FUNCTION_BLOCK PIDBase_HMI (* Service Interface Function Block Type *)
  (* Standard: 61499-2 *)
  (* Version 1.0.1, 10/18/2023, ApplicationLibDevTeam, Schneider Electric, First Version *)
  PACKAGE Main;
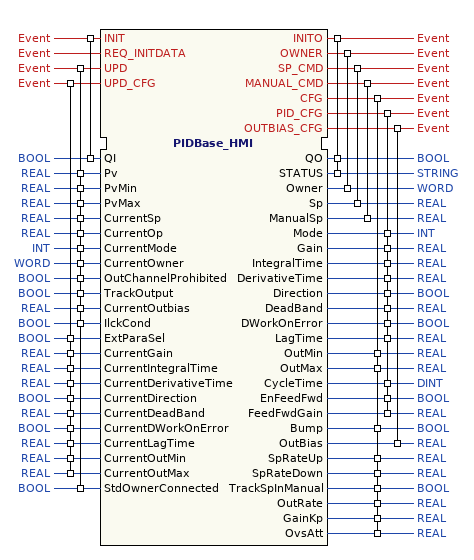
  EVENT_INPUT
    INIT WITH QI;
    REQ_INITDATA; (* Request to initialize data *)
    UPD WITH Pv, PvMin, PvMax, CurrentSp, CurrentOp, CurrentMode, OutChannelProhibited, TrackOutput, CurrentOutbias, IlckCond, StdOwnerConnected, CurrentOwner; (* Update data to supervision *)
    UPD_CFG WITH ExtParaSel, CurrentGain, CurrentIntegralTime, CurrentDerivativeTime, CurrentLagTime, CurrentDeadBand, CurrentOutMin, CurrentOutMax, CurrentDWorkOnError, CurrentDirection; (* Update external parameter data to supervision *)
  END_EVENT
  EVENT_OUTPUT
    INITO WITH QO, STATUS;
    OWNER WITH Owner; (* Request for owner change *)
    SP_CMD WITH Sp; (* Request to update operator setpoint in auto mode *)
    MANUAL_CMD WITH ManualSp; (* Request to update operator setpoint in manual mode *)
    CFG WITH OutMin, OutMax, Bump, SpRateUp, SpRateDown, TrackSpInManual, OutRate, GainKp, OvsAtt; (* Request to update generic parameters *)
    PID_CFG WITH Gain, DerivativeTime, IntegralTime, Mode, LagTime, DeadBand, Direction, CycleTime, DWorkOnError, EnFeedFwd, FeedFwdGain; (* Request to update PID parameter *)
    OUTBIAS_CFG WITH OutBias; (* Request to update outbias configuration *)
  END_EVENT
  VAR_INPUT
    QI : BOOL;
    Pv : REAL; (* Process value *) {SET_ATTRIBUTE(Runtime.Archive.Counters, AbsoluteValues=False)} {SET_ATTRIBUTE(Runtime.Archive.Id, 1)} {SET_ATTRIBUTE(Runtime.History.Depth, 500)} {SET_ATTRIBUTE(Runtime.History.SmoothTime, 60000)} {SET_ATTRIBUTE(Runtime.History.SmoothValue, 0.1)}
    PvMin : REAL; (* Minimum range of process value *)
    PvMax : REAL; (* Maximum range of process value *)
    CurrentSp : REAL; (* Current setpoint value *) {SET_ATTRIBUTE(Runtime.Archive.Counters, AbsoluteValues=False)} {SET_ATTRIBUTE(Runtime.Archive.Id, 1)} {SET_ATTRIBUTE(Runtime.History.Depth, 500)} {SET_ATTRIBUTE(Runtime.History.SmoothTime, 60000)} {SET_ATTRIBUTE(Runtime.History.SmoothValue, 0.1)}
    CurrentOp : REAL; (* Current output value *) {SET_ATTRIBUTE(Runtime.Archive.Counters, AbsoluteValues=False)} {SET_ATTRIBUTE(Runtime.Archive.Id, 1)} {SET_ATTRIBUTE(Runtime.History.Depth, 500)} {SET_ATTRIBUTE(Runtime.History.SmoothTime, 60000)} {SET_ATTRIBUTE(Runtime.History.SmoothValue, 0.1)}
    CurrentMode : INT; (* Current mode selected *)
    CurrentOwner : WORD; (* Current Owner status *)
    OutChannelProhibited : BOOL; (* 1 = Output change prohibited *)
    TrackOutput : BOOL; (* 1 = Output tracking active *)
    CurrentOutbias : REAL; (* Current ouput bias value *)
    IlckCond : BOOL; (* 1= Interlock active *)
    ExtParaSel : BOOL; (* 1 = External paramters available for PID calculation *)
    CurrentGain : REAL; (* Current gain for PID calculation *)
    CurrentIntegralTime : REAL; (* Current integral time for PID calculation *)
    CurrentDerivativeTime : REAL; (* Current derivative time for PID calculation *)
    CurrentDirection : BOOL; (* Current direction of PID calculation *)
    CurrentDeadBand : REAL; (* Current deadband for PID calculation *)
    CurrentDWorkOnError : BOOL; (* Current derivative work on error for PID calculation *)
    CurrentLagTime : REAL; (* Current lagtime for PID calculation *)
    CurrentOutMin : REAL; (* Current minimum ouput value for PID calculation *)
    CurrentOutMax : REAL; (* Current maximum ouput value for PID calculation *)
    StdOwnerConnected : BOOL; (* 1= External owner connected *)
  END_VAR
  VAR_OUTPUT
    QO : BOOL; (* Event Output Qualifier *)
    STATUS : STRING; (* Service Status *)
    Owner : WORD; (* Requested owner (16#10 = Operator, 16#8 = Program remote) *)
    Sp : REAL; (* Setpoint for PID calculation *)
    ManualSp : REAL; (* Manual setpoint for PID calculation *)
    Mode : INT; (* Mode for PID calculation (0 = Manual Mode, 1 = Auto Mode) *)
    Gain : REAL; (* Gain parameter for P calculation *)
    IntegralTime : REAL; (* Gain parameter for I calculation *)
    DerivativeTime : REAL; (* Parameter for D calculation *)
    Direction : BOOL; (* Direction for error calculation (0 = Pv-Sp; 1 = Sp-Pv) *)
    DeadBand : REAL; (* Deadband for I and D calculation *)
    DWorkOnError : BOOL; (* 1 = D work on error; 0 = D work on Pv *)
    LagTime : REAL; (* Lag time parameter for D calculation *)
    OutMin : REAL; (* Minimum range of ouput value *)
    OutMax : REAL; (* Maximum range of ouput value *)
    CycleTime : DINT; (* Cycletime for PID calculation (ms) *)
    EnFeedFwd : BOOL; (* 1 = Feedforward active *)
    FeedFwdGain : REAL; (* Feed forward gain value *)
    Bump : BOOL; (* 1 =Transition to automatic mode with bump ,0= Bumpless transition to automatic mode *)
    OutBias : REAL; (* Output offset (bias) value in Auto Mode and Integration time is zero *)
    SpRateUp : REAL; (* Setpoint rate to move up *)
    SpRateDown : REAL; (* Setpoint rate to move down *)
    TrackSpInManual : BOOL; (* 1 = Sp tracking to Pv is enabled in manual mode *)
    OutRate : REAL; (* Limit for output modification in units per second (≥ 0) *)
    GainKp : REAL; (* Reducing the proportional contribution within the dead zone dband *)
    OvsAtt : REAL; (* Reducing the overrun ( Should be between 0  to 1) *)
  END_VAR
  SERVICE /
    SEQUENCE 
    END_SEQUENCE
  END_SERVICE
END_FUNCTION_BLOCK
